// Brief: Calibrate the zero position of Instrument
FUNCTION_BLOCK PUBLIC FB_SlaveCtrlInstruCali EXTENDS FB_SlaveArmCtrlBase
VAR
	// flag to start calibration
	m_instruCaliStart:BOOL;
	
	// mount motion planning
	m_jntOTG :ARRAY[1..8] OF FB_secOrdTrajFilter;
	m_instruMountVel :LREAL := 1*PI;
	m_instruMountAcc :LREAL := 2*PI;
	
	// 	cali status
	m_rollJntCaliStatus :INT := 0;
	m_pitchJntCaliStatus :INT := 0;
	m_yawJntCaliStatus :INT := 0;
	
	// flag if zero position is written to CoE
	m_zeroPosWritten :BOOL;
	m_zeroPosWriteStart :BOOL;
	
	// flag if SN is written to CoE
	m_SNWritten:BOOL;
	m_SNWriteStart:BOOL;
	
	// joint current threshold which indicate panel is buckled with instrument
	m_maxJntCurrent :LREAL := 100;
	
	// joint current threshold which indicate finger closed
	m_fingerCloseCurrent :LREAL := 50;
	
	// joint position at limits
	m_jntLimitPos1, m_jntLimitPos2, m_jntCaliPos :LREAL;
	m_jntLimitPos3, m_jntLimitPos4 :LREAL;

	// flag if joint is mounted
	m_jointMounted :ARRAY[1..8] OF BOOL := [5(FALSE)];
	
	// instrument mount motion range
	m_mountMotionAng :LREAL :=30*g_deg2Rad;
	
	// command mount motion
	m_targetMountPos :Vec8d;
	
	// instrument zero position
	m_instruZeroPosition :Vec5d;
	
	// angle to close finger
	m_baseCloseAngle :LREAL := 1*g_deg2Rad;
	m_bipolarCloseAngle :LREAL := 5*g_deg2Rad;
	m_proGraspCloseAngle:LREAL := 25*g_deg2Rad;
	
END_VAR

// override this function in each exact controller
METHOD PROTECTED calcCmdJntPos : BOOL
VAR_IN_OUT CONSTANT
	i_endoscopePose : ST_Frame;
	i_masterStatus :ST_MasterStatus;
	i_setupStatus: ST_SetupStatus;
	i_slaveArm :FB_SlaveArm;
END_VAR

VAR 
	i :INT;
END_VAR
// retur directly if instrument/endoscope is not readed
IF NOT i_slaveArm.instrument.onChipData.m_InstruReadSucceed THEN
	m_rollJntCaliStatus :=0;
	m_pitchJntCaliStatus :=0;
	m_yawJntCaliStatus :=0;
	m_zeroPosWritten :=FALSE;
	m_zeroPosWriteStart:=FALSE;
	m_SNWritten :=FALSE;
	m_SNWriteStart:=FALSE;
	m_instruCaliStart:=FALSE;
	FOR i:=4 TO 8 DO
		m_jointMounted[i]:=FALSE;
	END_FOR
	return;
END_IF

// write SN to CoE
IF GVL_InstruTestUIVars.g_writeSNFlag THEN
	m_SNWriteStart := TRUE;
ELSE
	IF m_SNWriteStart THEN
		IF   NOT m_SNWritten THEN
			m_SNWritten := i_slaveArm.instrument.writeSNToChip(GVL_InstruTestUIVars.g_newInstruSN);
		ELSE
			m_SNWriteStart :=FALSE;
			m_SNWritten:=FALSE;
		END_IF
	END_IF
END_IF

// write zero position to CoE
IF GVL_InstruTestUIVars.g_writeZeroPosFlag THEN
	m_zeroPosWriteStart := TRUE;
ELSE
	IF m_yawJntCaliStatus = -1 AND m_zeroPosWriteStart THEN
		IF   NOT m_zeroPosWritten THEN
			m_zeroPosWritten := i_slaveArm.instrument.writeZeroPosToChip(m_instruZeroPosition[1],m_instruZeroPosition[2],m_instruZeroPosition[3]);	
		ELSE
			m_zeroPosWriteStart:=FALSE;
			m_zeroPosWritten:=FALSE;
		END_IF
		RETURN;
	END_IF;
END_IF


// move joint to zero position
IF GVL_InstruTestUIVars.g_searchZeroPosFlag THEN
	m_rollJntCaliStatus :=0;
	m_pitchJntCaliStatus :=0;
	m_yawJntCaliStatus :=0;
	m_instruCaliStart := TRUE;
ELSE
	IF m_instruCaliStart THEN
		// calibrate motion
		IF m_rollJntCaliStatus <> -1 THEN
			rollJntCali(i_slaveArm);
		ELSIF m_pitchJntCaliStatus <> -1 THEN
			pitchJntCali(i_slaveArm);
		ELSIF m_yawJntCaliStatus <> -1 THEN
			IF  i_slaveArm.instrument.instruTypeInfo.m_isSingleFinger THEN
				yawJntCali_finger(i_slaveArm);
			ELSE
				yawJntCali_gripper(i_slaveArm);
			END_IF
		
		END_IF
		
		// calibrate motion finish and record position
		IF m_yawJntCaliStatus = -1 THEN
			FOR  i:=1 TO  5 DO
				m_instruZeroPosition[i]:=i_slaveArm.linkSingle[i+3];
			END_FOR
			m_instruCaliStart:=FALSE;
		END_IF
	END_IF
		
END_IF
END_METHOD

METHOD PUBLIC init : BOOL
VAR_IN_OUT CONSTANT
	i_slaveArm	:FB_SlaveArm;
END_VAR
VAR_IN_OUT 
	r_slaveArmCtrlCmd :ST_SlaveArmCtrlCmds;
END_VAR

VAR
	i : INT;
END_VAR
// check if to hold the command joint position unchanged
m_holdLastCmds := checkToHoldLastCmds(i_slaveArm);

SUPER^.Init(i_slaveArm,r_slaveArmCtrlCmd);
m_jntOPMode[4] := DriverOPMode_PosTrq;
m_jntOPMode[5] := DriverOPMode_PosTrq;
m_jntOPMode[6] := DriverOPMode_PosTrq;
m_jntOPMode[7] := DriverOPMode_PosTrq;
m_jntOPMode[8] := DriverOPMode_PosTrq;

FOR i:=4 TO 8 DO
	m_targetMountPos[i]:=m_cmdJntPos[i];
	m_jntOTG[i].init(m_targetMountPos[i], 0,m_instruMountVel, m_instruMountAcc, g_slaveArmCtrlCycleTime);
	m_jointMounted[i]:=FALSE;
END_FOR

m_rollJntCaliStatus :=0;
m_pitchJntCaliStatus :=0;
m_yawJntCaliStatus :=0;
m_zeroPosWritten := FALSE;

m_zeroPosWriteStart:=FALSE;
m_SNWritten :=FALSE;
m_SNWriteStart:=FALSE;
m_instruCaliStart:=FALSE;

// update commands to arm
copyCmds(r_slaveArmCtrlCmd);
END_METHOD

METHOD pitchJntCali : BOOL
VAR_IN_OUT CONSTANT
	i_slaveArm :FB_SlaveArm;
END_VAR

VAR 
	i :INT;
	curJntPos :Vec8d;
	jntIdx :INT;
END_VAR
jntIdx:=6;
curJntPos := i_slaveArm.curJntPos;

CASE m_pitchJntCaliStatus OF
	// rotate clockwise
	0:
		m_targetMountPos[jntIdx]:=curJntPos[jntIdx]+m_mountMotionAng;
	
		//buckle joint
		IF i_slaveArm.filtJntCurrent[jntIdx]> m_maxJntCurrent THEN 
			m_jntLimitPos1 := curJntPos[jntIdx];
			m_targetMountPos[jntIdx]:=curJntPos[jntIdx];
			m_jntOTG[jntIdx].init(m_targetMountPos[jntIdx], 0,m_instruMountVel, m_instruMountAcc, g_slaveArmCtrlCycleTime);
			m_pitchJntCaliStatus := 1;
		END_IF
		
	// rotate anticlockwise
	1:
		m_targetMountPos[jntIdx]:=curJntPos[jntIdx]-m_mountMotionAng;
	
		//buckle  joint
		IF i_slaveArm.filtJntCurrent[jntIdx]<- m_maxJntCurrent THEN 
			m_jntLimitPos2 := curJntPos[jntIdx];
			m_targetMountPos[jntIdx]:=curJntPos[jntIdx];
			m_jntOTG[jntIdx].init(m_targetMountPos[jntIdx], 0,m_instruMountVel, m_instruMountAcc, g_slaveArmCtrlCycleTime);
			m_pitchJntCaliStatus := 2;
		END_IF
	
	2:// calculate center/calibarted position
		m_targetMountPos[jntIdx] :=  (m_jntLimitPos1 + m_jntLimitPos2)/2+ i_slaveArm.instrument.instruTypeInfo.m_instruPitchBachlash/2.0;
		m_pitchJntCaliStatus := 3;

	3:
		IF ABS(m_targetMountPos[jntIdx]-curJntPos[jntIdx]) <GVL_SlaveControlParameters.g_jntCtrlAngTolHigh  THEN
			m_pitchJntCaliStatus := -1;
		END_IF
		
END_CASE

// traj plan
m_jntOTG[jntIdx].run(m_targetMountPos[jntIdx],0.0, o_cmdAcc=>m_cmdJntAcc[jntIdx],o_cmdVel=>m_cmdJntVel[jntIdx],o_cmdPos=>m_cmdJntPos[jntIdx]);
END_METHOD

METHOD rollJntCali : BOOL
VAR_IN_OUT CONSTANT
	i_slaveArm :FB_SlaveArm;
END_VAR

VAR 
	i :INT;
	curJntPos :Vec8d;
	jntIdx :INT;
END_VAR
jntIdx:=7;
curJntPos := i_slaveArm.curJntPos;

CASE m_rollJntCaliStatus OF
	// rotate clockwise
	0:
		m_targetMountPos[jntIdx]:=curJntPos[jntIdx]+m_mountMotionAng;
	
		//buckle  joint
		IF i_slaveArm.filtJntCurrent[jntIdx]> m_maxJntCurrent AND ABS(i_slaveArm.curJntVel[jntIdx]) < 1*g_deg2rad  THEN 
			m_jntLimitPos1 := curJntPos[jntIdx];
			m_targetMountPos[jntIdx]:=curJntPos[jntIdx];
			m_jntOTG[jntIdx].init(m_targetMountPos[jntIdx], 0,m_instruMountVel, m_instruMountAcc, g_slaveArmCtrlCycleTime);
			m_rollJntCaliStatus := 1;
		END_IF
		
	// rotate anticlockwise
	1:
		m_targetMountPos[jntIdx]:=curJntPos[jntIdx]-m_mountMotionAng;
	
		//buckle  joint
		IF i_slaveArm.filtJntCurrent[jntIdx]<- m_maxJntCurrent AND ABS(i_slaveArm.curJntVel[jntIdx]) < 1*g_deg2rad   THEN 
			m_jntLimitPos2 := curJntPos[jntIdx];
			m_targetMountPos[jntIdx]:=curJntPos[jntIdx];
			m_jntOTG[jntIdx].init(m_targetMountPos[jntIdx], 0,m_instruMountVel, m_instruMountAcc, g_slaveArmCtrlCycleTime);
			m_rollJntCaliStatus := 2;
		END_IF
	
	2:// calculate center/calibarted positio
		m_targetMountPos[jntIdx] :=  (m_jntLimitPos1 + m_jntLimitPos2)/2;
		m_rollJntCaliStatus := 3;

	3:
		IF ABS(m_targetMountPos[jntIdx]-curJntPos[jntIdx]) <GVL_SlaveControlParameters.g_jntCtrlAngTolHigh  THEN
			m_rollJntCaliStatus := -1;
		END_IF
		
END_CASE

// traj plan
m_jntOTG[jntIdx].run(m_targetMountPos[jntIdx],0.0, o_cmdAcc=>m_cmdJntAcc[jntIdx],o_cmdVel=>m_cmdJntVel[jntIdx],o_cmdPos=>m_cmdJntPos[jntIdx]);
END_METHOD

METHOD yawJntCali_finger : BOOL
VAR_IN_OUT CONSTANT
	i_slaveArm :FB_SlaveArm;
END_VAR

VAR 
	i :INT;
	curJntPos :Vec8d;
	jntIdx :INT;
END_VAR
jntIdx:=5;
curJntPos := i_slaveArm.curJntPos;

CASE m_yawJntCaliStatus OF
	// rotate clockwise
	0:
		m_targetMountPos[jntIdx]:=curJntPos[jntIdx]+m_mountMotionAng;
	
		//buckle  joint
		IF i_slaveArm.filtJntCurrent[jntIdx]> m_maxJntCurrent THEN 
			m_jntLimitPos1 := curJntPos[jntIdx];
			m_targetMountPos[jntIdx]:=curJntPos[jntIdx];
			m_jntOTG[jntIdx].init(m_targetMountPos[jntIdx], 0,m_instruMountVel, m_instruMountAcc, g_slaveArmCtrlCycleTime);
			m_yawJntCaliStatus := 1;
		END_IF
		
	// rotate anticlockwise
	1:
		m_targetMountPos[jntIdx]:=curJntPos[jntIdx]-m_mountMotionAng;
	
		//buckle  joint
		IF i_slaveArm.filtJntCurrent[jntIdx]<- m_maxJntCurrent THEN 
			m_jntLimitPos2 := curJntPos[jntIdx];
			m_targetMountPos[jntIdx]:=curJntPos[jntIdx];
			m_jntOTG[jntIdx].init(m_targetMountPos[jntIdx], 0,m_instruMountVel, m_instruMountAcc, g_slaveArmCtrlCycleTime);
			m_yawJntCaliStatus := 2;
		END_IF
	
	2:// calculate center/calibarted positio
		m_targetMountPos[jntIdx] :=  (m_jntLimitPos1 + m_jntLimitPos2)/2+i_slaveArm.instrument.instruTypeInfo.m_instruYawBacklash/2.0;;
		m_yawJntCaliStatus := 3;

	3:
		IF ABS(m_targetMountPos[jntIdx]-curJntPos[jntIdx]) <GVL_SlaveControlParameters.g_jntCtrlAngTolLow  THEN
			m_yawJntCaliStatus := -1;
		END_IF
		
END_CASE

// traj plan
m_jntOTG[jntIdx].run(m_targetMountPos[jntIdx],0.0, o_cmdAcc=>m_cmdJntAcc[jntIdx],o_cmdVel=>m_cmdJntVel[jntIdx],o_cmdPos=>m_cmdJntPos[jntIdx]);
END_METHOD

METHOD yawJntCali_gripper : BOOL
VAR_IN_OUT CONSTANT
	i_slaveArm :FB_SlaveArm;
END_VAR

VAR 
	curJntPos :Vec8d;
	gripCloseAng:LREAL;
END_VAR
curJntPos := i_slaveArm.curJntPos;

// determin finger close angle
IF i_slaveArm.instrument.instruType = InstruType_MarylandForceps OR i_slaveArm.instrument.instruType = InstruType_FenestratedForceps
	OR i_slaveArm.instrument.instruType = InstruType_CurvedBipolarDissector OR i_slaveArm.instrument.instruType = InstruType_MicroBipolarForceps THEN
	gripCloseAng := m_bipolarCloseAngle;
ELSIF i_slaveArm.instrument.instruType = InstruType_ProGraspForceps OR i_slaveArm.instrument.instruType = InstruType_ForceBipolar THEN
	gripCloseAng := m_proGraspCloseAngle;
ELSE
	gripCloseAng := m_baseCloseAngle;
END_IF

CASE m_yawJntCaliStatus OF
	// buckle joint4 and joint5 by moving toward limit
	0:
		//buckle panel with instrument
		// check if buckled 
		IF i_slaveArm.filtJntCurrent[4]<- m_maxJntCurrent THEN 
			m_jointMounted[4]:=TRUE;
			m_targetMountPos[4]:=curJntPos[4];
			m_jntOTG[4].init(m_targetMountPos[4], 0,m_instruMountVel, m_instruMountAcc, g_slaveArmCtrlCycleTime);
		END_IF
		IF i_slaveArm.filtJntCurrent[5]<- m_maxJntCurrent THEN 
			m_jointMounted[5]:=TRUE;
			m_targetMountPos[5]:=curJntPos[5];
			m_jntOTG[5].init(m_targetMountPos[5], 0,m_instruMountVel, m_instruMountAcc, g_slaveArmCtrlCycleTime);
		END_IF
		
		// set target joint position
		IF FALSE = m_jointMounted[4] THEN
			m_targetMountPos[4]:=curJntPos[4]-m_mountMotionAng;
		END_IF
		IF FALSE = m_jointMounted[5] THEN
			m_targetMountPos[5]:=curJntPos[5]-m_mountMotionAng;
		END_IF

		IF m_jointMounted[4] AND m_jointMounted[5] THEN
			m_yawJntCaliStatus := 1;
			m_jointMounted[4]:=FALSE;
			m_jointMounted[5]:=FALSE;
		END_IF
	// close finger
	1:
		//buckle panel with instrument
		// check if buckled 
		IF i_slaveArm.filtJntCurrent[4]> m_maxJntCurrent THEN 
			m_jointMounted[4]:=TRUE;
			m_targetMountPos[4]:=curJntPos[4];
			m_jntOTG[4].init(m_targetMountPos[4], 0,m_instruMountVel, m_instruMountAcc, g_slaveArmCtrlCycleTime);
		END_IF
		IF i_slaveArm.filtJntCurrent[5]> m_maxJntCurrent THEN 
			m_jointMounted[5]:=TRUE;
			m_targetMountPos[5]:=curJntPos[5];
			m_jntOTG[5].init(m_targetMountPos[5], 0,m_instruMountVel, m_instruMountAcc, g_slaveArmCtrlCycleTime);
		END_IF
		
		// set target joint position
		IF FALSE = m_jointMounted[4] THEN
			m_targetMountPos[4]:=curJntPos[4]+m_mountMotionAng;
		END_IF
		IF FALSE = m_jointMounted[5] THEN
			m_targetMountPos[5]:=curJntPos[5]+m_mountMotionAng;
		END_IF

		IF m_jointMounted[4] AND m_jointMounted[5] THEN
			m_yawJntCaliStatus := 2;
			m_jointMounted[4]:=FALSE;
			m_jointMounted[5]:=FALSE;
		END_IF
		
	2:// move joint5 to open gripper
		m_targetMountPos[4] := curJntPos[4]-i_slaveArm.instrument.instruTypeInfo.m_maxGripAngle/4.0;
		m_targetMountPos[5] := curJntPos[5]-i_slaveArm.instrument.instruTypeInfo.m_maxGripAngle/4.0;
		m_yawJntCaliStatus := 3;

	3:
		IF ABS(m_targetMountPos[5]-curJntPos[5]) <GVL_SlaveControlParameters.g_jntCtrlAngTolLow  THEN
			m_yawJntCaliStatus := 4;
		END_IF
			
	// roll clockwise to reach limit
	4:
		IF NOT(m_jointMounted[4]) THEN  
			// set target joint position
			m_targetMountPos[4]:=curJntPos[4]-m_mountMotionAng;
			// check if reach limit 
			IF i_slaveArm.filtJntCurrent[4]< -m_maxJntCurrent THEN 
				m_jointMounted[4]:=TRUE;
				m_jntLimitPos1 := curJntPos[4];
				m_targetMountPos[4]:=curJntPos[4];
				m_jntOTG[4].init(m_targetMountPos[4], 0,m_instruMountVel, m_instruMountAcc, g_slaveArmCtrlCycleTime);
			END_IF
		END_IF
		IF NOT(m_jointMounted[5]) THEN 
			// set target joint position
			m_targetMountPos[5]:=curJntPos[5]+m_mountMotionAng;
			// check if reach limit 
			IF i_slaveArm.filtJntCurrent[5]> m_maxJntCurrent THEN 
				m_jointMounted[5]:=TRUE;
				m_jntLimitPos2 := curJntPos[5];
				m_targetMountPos[5]:=curJntPos[5];
				m_jntOTG[5].init(m_targetMountPos[5], 0,m_instruMountVel, m_instruMountAcc, g_slaveArmCtrlCycleTime);
			END_IF	
		END_IF
		
		// transit
		IF m_jointMounted[4] AND m_jointMounted[5] THEN
			m_yawJntCaliStatus := 5;
			m_jointMounted[4]:=FALSE;
			m_jointMounted[5]:= FALSE;
		END_IF
		
	5:// move joint5 to open gripper
		m_targetMountPos[5] := curJntPos[5]-i_slaveArm.instrument.instruTypeInfo.m_maxGripAngle/2.0;
		m_yawJntCaliStatus := 6;

	6:
		IF ABS(m_targetMountPos[5]-curJntPos[5]) <GVL_SlaveControlParameters.g_jntCtrlAngTolLow  THEN
			m_yawJntCaliStatus := 7;
		END_IF

	// roll anticlockwise to reach limit
	7:
		IF NOT(m_jointMounted[4]) THEN  
			// set target joint position
			m_targetMountPos[4]:=curJntPos[4]+m_mountMotionAng;
			// check if reach limit 
			IF i_slaveArm.filtJntCurrent[4]>m_maxJntCurrent THEN 
				m_jointMounted[4]:=TRUE;
				m_jntLimitPos3 := curJntPos[4];
				m_targetMountPos[4]:=curJntPos[4];
				m_jntOTG[4].init(m_targetMountPos[4], 0,m_instruMountVel, m_instruMountAcc, g_slaveArmCtrlCycleTime);
			END_IF
		END_IF
		IF NOT(m_jointMounted[5]) THEN 
			// set target joint position
			m_targetMountPos[5]:=curJntPos[5]-m_mountMotionAng;
			// check if reach limit 
			IF i_slaveArm.filtJntCurrent[5]<- m_maxJntCurrent THEN 
				m_jointMounted[5]:=TRUE;
				m_jntLimitPos4 := curJntPos[5];
				m_targetMountPos[5]:=curJntPos[5];
				m_jntOTG[5].init(m_targetMountPos[5], 0,m_instruMountVel, m_instruMountAcc, g_slaveArmCtrlCycleTime);
			END_IF	
		END_IF
		
		// transit
		IF m_jointMounted[4] AND m_jointMounted[5] THEN
			m_yawJntCaliStatus := 8;
			m_jointMounted[4]:=FALSE;
			m_jointMounted[5]:= FALSE;
		END_IF
		
	8:// calculate center/calibarted position
		m_targetMountPos[4] := (m_jntLimitPos1 + m_jntLimitPos3)/2-i_slaveArm.instrument.instruTypeInfo.m_instruYawBacklash/2.0;
		m_targetMountPos[5] := (m_jntLimitPos2 + m_jntLimitPos4)/2+i_slaveArm.instrument.instruTypeInfo.m_instruYawBacklash/2.0;
		m_yawJntCaliStatus := 9;

	9:
		IF ABS(m_targetMountPos[4]-curJntPos[4]) <GVL_SlaveControlParameters.g_jntCtrlAngTolLow  AND
			ABS(m_targetMountPos[5]-curJntPos[5]) <GVL_SlaveControlParameters.g_jntCtrlAngTolLow  THEN
			m_targetMountPos[4] := curJntPos[4]+i_slaveArm.instrument.instruTypeInfo.m_instruYawBacklash;
			m_yawJntCaliStatus := 10;
		END_IF
		
	// close finger	
	10:
		IF ABS(m_targetMountPos[4]-curJntPos[4]) <GVL_SlaveControlParameters.g_jntCtrlAngTolLow  AND
			ABS(m_targetMountPos[5]-curJntPos[5]) <GVL_SlaveControlParameters.g_jntCtrlAngTolLow  THEN
				m_targetMountPos[4] := curJntPos[4]+gripCloseAng;
				m_targetMountPos[5] := curJntPos[5]+gripCloseAng;
			m_yawJntCaliStatus := 11;
		END_IF
		

	11:
		IF ABS(m_targetMountPos[4]-curJntPos[4]) <GVL_SlaveControlParameters.g_jntCtrlAngTolLow  AND
			ABS(m_targetMountPos[5]-curJntPos[5]) <GVL_SlaveControlParameters.g_jntCtrlAngTolLow  THEN
			m_yawJntCaliStatus := -1;
		END_IF

END_CASE

// traj plan
m_jntOTG[4].run(m_targetMountPos[4],0.0, o_cmdAcc=>m_cmdJntAcc[4],o_cmdVel=>m_cmdJntVel[4],o_cmdPos=>m_cmdJntPos[4]);
m_jntOTG[5].run(m_targetMountPos[5],0.0, o_cmdAcc=>m_cmdJntAcc[5],o_cmdVel=>m_cmdJntVel[5],o_cmdPos=>m_cmdJntPos[5]);
END_METHOD

END_FUNCTION_BLOCK

(* stored: Version 1.1.0.1, ProductVersion 3.1.4024.12
   POU FB_SlaveCtrlInstruCali: Id {f6122a4e-e5d8-4252-8b12-6598a16e0174}, SpecialFunc None
   Method calcCmdJntPos: Id {92420bbe-f9a2-4f31-a213-0e60613d7858}
   Method init: Id {d75d663d-308e-4f56-ae72-9d04b2f0e2be}
   Method pitchJntCali: Id {e9c6d1cd-4c78-4bd5-b668-b8facd8b1f86}
   Method rollJntCali: Id {6fecbb26-dee3-460d-8ebc-c5e9758738f5}
   Method yawJntCali_finger: Id {367337ae-1143-4558-b119-2ddaf442a22f}
   Method yawJntCali_gripper: Id {98a7face-4e61-461c-9585-b9ec777fc235} *)
